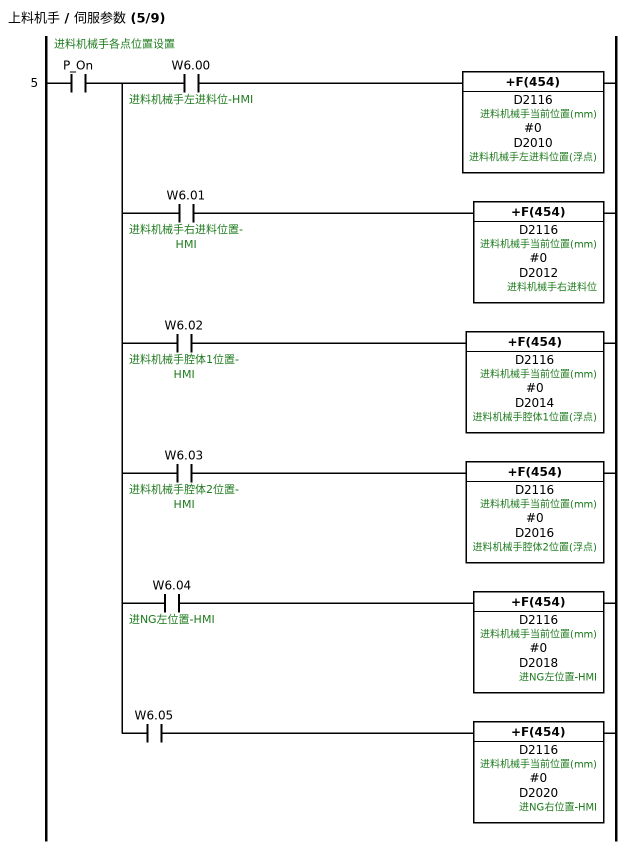
; [picture p96: 上料机手 / 伺服参数, rungs 5-5]
; rung 5: 进料机械手各点位置设置
LD P_On
OUT TR0
AND W6.00  ; 进料机械手左进料位-HMI
+F(454) D2116 #0 D2010  ; 进料机械手当前位置(mm), 进料机械手左进料位置(浮点)
LD TR0
AND W6.01  ; 进料机械手右进料位置-HMI
+F(454) D2116 #0 D2012  ; 进料机械手当前位置(mm), 进料机械手右进料位
LD TR0
AND W6.02  ; 进料机械手腔体1位置-HMI
+F(454) D2116 #0 D2014  ; 进料机械手当前位置(mm), 进料机械手腔体1位置(浮点)
LD TR0
AND W6.03  ; 进料机械手腔体2位置-HMI
+F(454) D2116 #0 D2016  ; 进料机械手当前位置(mm), 进料机械手腔体2位置(浮点)
LD TR0
AND W6.04  ; 进NG左位置-HMI
+F(454) D2116 #0 D2018  ; 进料机械手当前位置(mm), 进NG左位置-HMI
LD TR0
AND W6.05
+F(454) D2116 #0 D2020  ; 进料机械手当前位置(mm), 进NG右位置-HMI

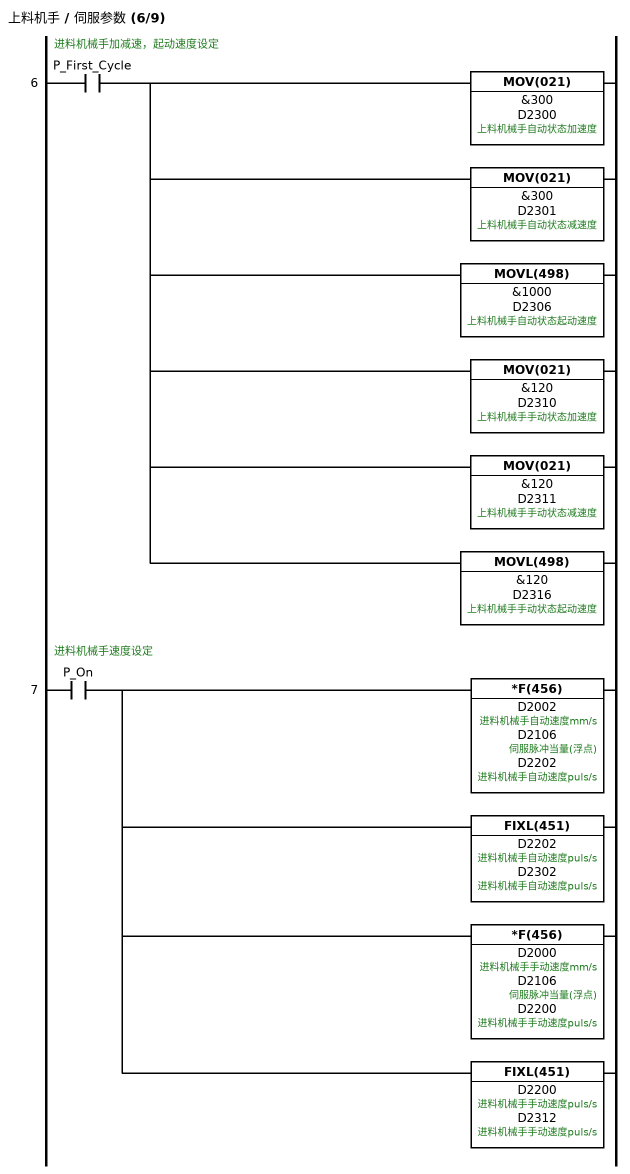
; rung 6: 进料机械手加减速，起动速度设定
LD P_First_Cycle
MOV(021) &300 D2300  ; 上料机械手自动状态加速度
MOV(021) &300 D2301  ; 上料机械手自动状态减速度
MOVL(498) &1000 D2306  ; 上料机械手自动状态起动速度
MOV(021) &120 D2310  ; 上料机械手手动状态加速度
MOV(021) &120 D2311  ; 上料机械手手动状态减速度
MOVL(498) &120 D2316  ; 上料机械手手动状态起动速度
; rung 7: 进料机械手速度设定
LD P_On
*F(456) D2002 D2106 D2202  ; 进料机械手自动速度mm/s, 伺服脉冲当量(浮点), 进料机械手自动速度puls/s
FIXL(451) D2202 D2302  ; 进料机械手自动速度puls/s
*F(456) D2000 D2106 D2200  ; 进料机械手手动速度mm/s, 伺服脉冲当量(浮点), 进料机械手手动速度puls/s
FIXL(451) D2200 D2312  ; 进料机械手手动速度puls/s

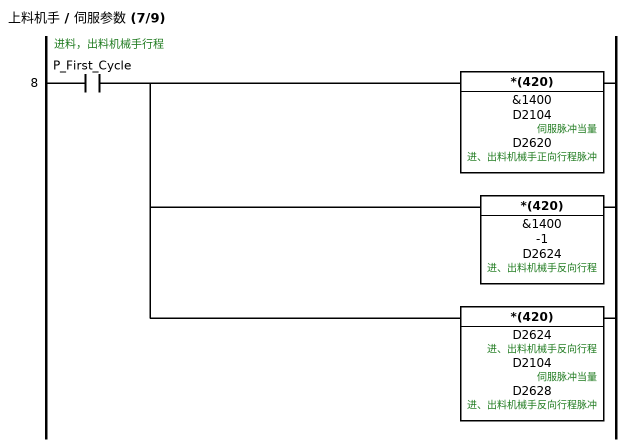
; rung 8: 进料，出料机械手行程
LD P_First_Cycle
*(420) &1400 D2104 D2620  ; 伺服脉冲当量, 进、出料机械手正向行程脉冲
*(420) &1400 -1 D2624  ; 进、出料机械手反向行程
*(420) D2624 D2104 D2628  ; 进、出料机械手反向行程, 伺服脉冲当量, 进、出料机械手反向行程脉冲

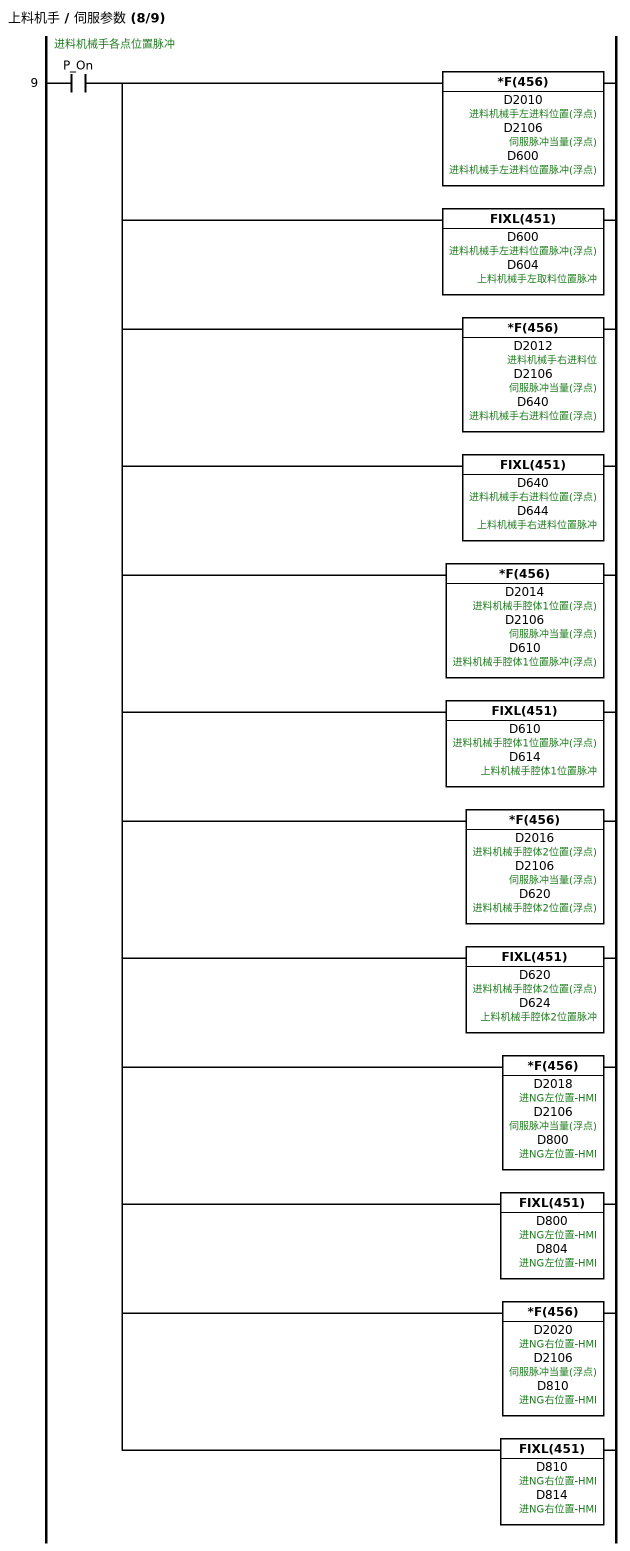
; rung 9: 进料机械手各点位置脉冲
LD P_On
*F(456) D2010 D2106 D600  ; 进料机械手左进料位置(浮点), 伺服脉冲当量(浮点), 进料机械手左进料位置脉冲(浮点)
FIXL(451) D600 D604  ; 进料机械手左进料位置脉冲(浮点), 上料机械手左取料位置脉冲
*F(456) D2012 D2106 D640  ; 进料机械手右进料位, 伺服脉冲当量(浮点), 进料机械手右进料位置(浮点)
FIXL(451) D640 D644  ; 进料机械手右进料位置(浮点), 上料机械手右进料位置脉冲
*F(456) D2014 D2106 D610  ; 进料机械手腔体1位置(浮点), 伺服脉冲当量(浮点), 进料机械手腔体1位置脉冲(浮点)
FIXL(451) D610 D614  ; 进料机械手腔体1位置脉冲(浮点), 上料机械手腔体1位置脉冲
*F(456) D2016 D2106 D620  ; 进料机械手腔体2位置(浮点), 伺服脉冲当量(浮点)
FIXL(451) D620 D624  ; 进料机械手腔体2位置(浮点), 上料机械手腔体2位置脉冲
*F(456) D2018 D2106 D800  ; 进NG左位置-HMI, 伺服脉冲当量(浮点)
FIXL(451) D800 D804  ; 进NG左位置-HMI
*F(456) D2020 D2106 D810  ; 进NG右位置-HMI, 伺服脉冲当量(浮点)
FIXL(451) D810 D814  ; 进NG右位置-HMI

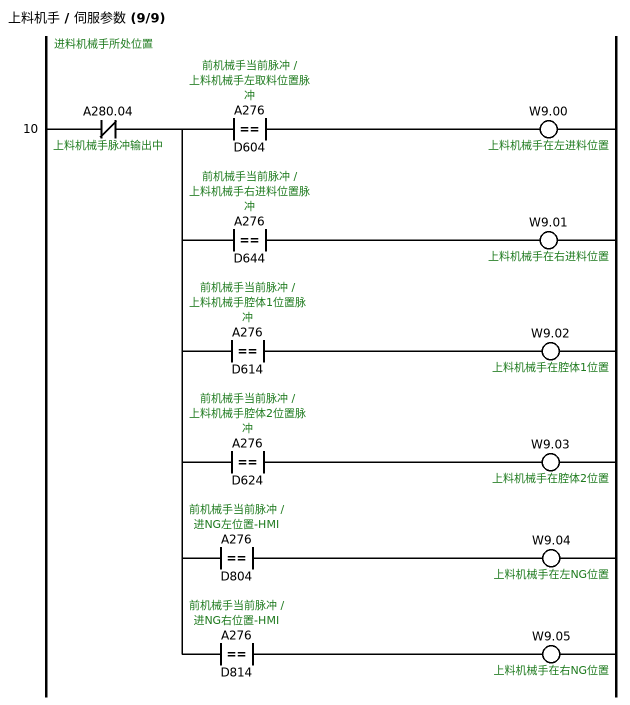
; rung 10: 进料机械手所处位置
LDNOT A280.04  ; 上料机械手脉冲输出中
OUT TR0
AND=SL(303) A276 D604  ; 前机械手当前脉冲, 上料机械手左取料位置脉冲
OUT W9.00  ; 上料机械手在左进料位置
LD TR0
AND=SL(303) A276 D644  ; 前机械手当前脉冲, 上料机械手右进料位置脉冲
OUT W9.01  ; 上料机械手在右进料位置
LD TR0
AND=SL(303) A276 D614  ; 前机械手当前脉冲, 上料机械手腔体1位置脉冲
OUT W9.02  ; 上料机械手在腔体1位置
LD TR0
AND=SL(303) A276 D624  ; 前机械手当前脉冲, 上料机械手腔体2位置脉冲
OUT W9.03  ; 上料机械手在腔体2位置
LD TR0
AND=SL(303) A276 D804  ; 前机械手当前脉冲, 进NG左位置-HMI
OUT W9.04  ; 上料机械手在左NG位置
LD TR0
AND=SL(303) A276 D814  ; 前机械手当前脉冲, 进NG右位置-HMI
OUT W9.05  ; 上料机械手在右NG位置

### Section 外部输出及轴控运动

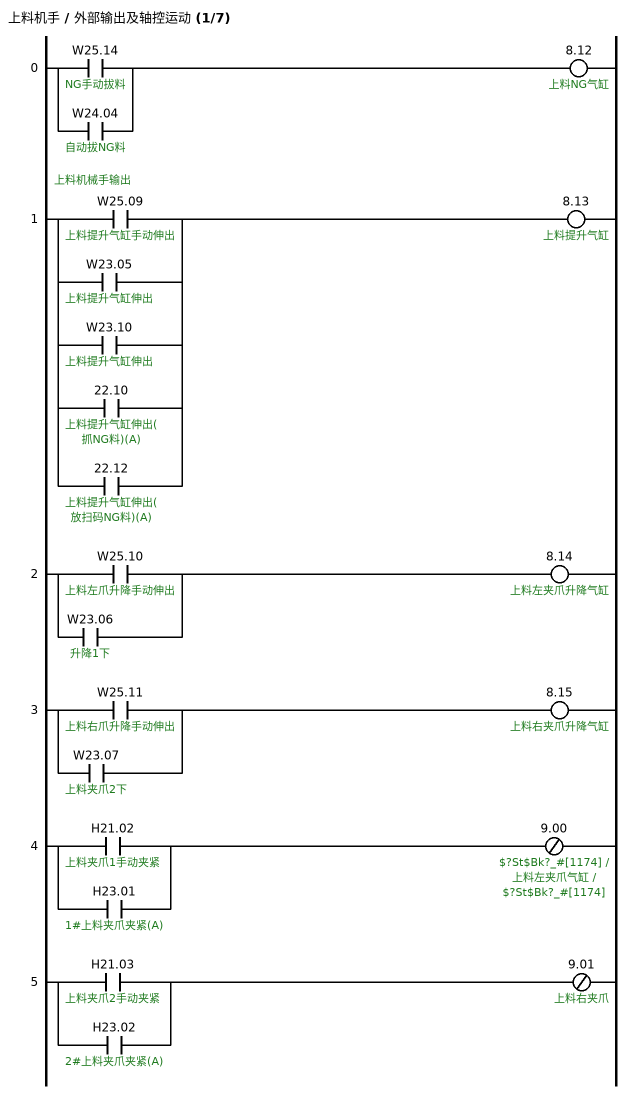
; rung 0
LD W25.14  ; NG手动拔料
OR W24.04  ; 自动拔NG料
OUT 8.12  ; 上料NG气缸
; rung 1: 上料机械手输出
LD W25.09  ; 上料提升气缸手动伸出
OR W23.05  ; 上料提升气缸伸出
OR W23.10  ; 上料提升气缸伸出
OR 22.10  ; 上料提升气缸伸出(抓NG料)(A)
OR 22.12  ; 上料提升气缸伸出(放扫码NG料)(A)
OUT 8.13  ; 上料提升气缸
; rung 2
LD W25.10  ; 上料左爪升降手动伸出
OR W23.06  ; 升降1下
OUT 8.14  ; 上料左夹爪升降气缸
; rung 3
LD W25.11  ; 上料右爪升降手动伸出
OR W23.07  ; 上料夹爪2下
OUT 8.15  ; 上料右夹爪升降气缸
; rung 4
LD H21.02  ; 上料夹爪1手动夹紧
OR H23.01  ; 1#上料夹爪夹紧(A)
OUTNOT 9.00  ; $?St$Bk?_#[1174] / 上料左夹爪气缸 / $?St$Bk?_#[1174]
; rung 5
LD H21.03  ; 上料夹爪2手动夹紧
OR H23.02  ; 2#上料夹爪夹紧(A)
OUTNOT 9.01  ; 上料右夹爪

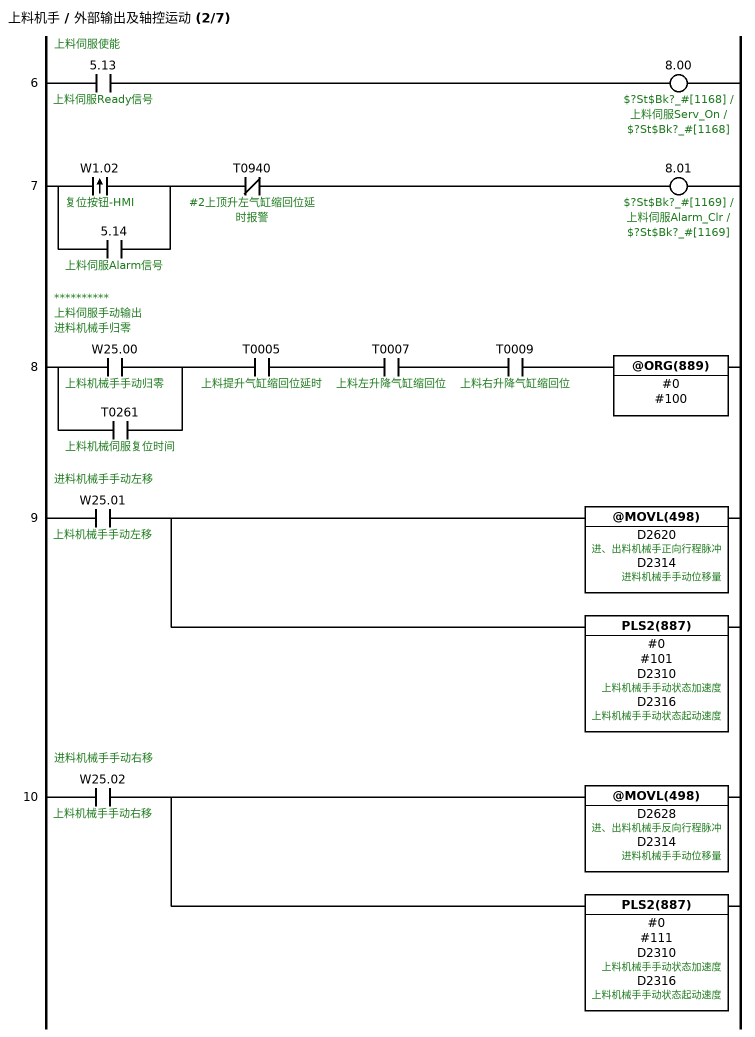
; rung 6: 上料伺服使能
LD 5.13  ; 上料伺服Ready信号
OUT 8.00  ; $?St$Bk?_#[1168] / 上料伺服Serv_On / $?St$Bk?_#[1168]
; rung 7
@LD W1.02  ; 复位按钮-HMI
OR 5.14  ; 上料伺服Alarm信号
ANDNOT T0940  ; #2上顶升左气缸缩回位延时报警
OUT 8.01  ; $?St$Bk?_#[1169] / 上料伺服Alarm_Clr / $?St$Bk?_#[1169]
; rung 8: ********** / 上料伺服手动输出 / 进料机械手归零
LD W25.00  ; 上料机械手手动归零
OR T0261  ; 上料机械伺服复位时间
AND T0005  ; 上料提升气缸缩回位延时
AND T0007  ; 上料左升降气缸缩回位
AND T0009  ; 上料右升降气缸缩回位
@ORG(889) #0 #100
; rung 9: 进料机械手手动左移
LD W25.01  ; 上料机械手手动左移
@MOVL(498) D2620 D2314  ; 进、出料机械手正向行程脉冲, 进料机械手手动位移量
PLS2(887) #0 #101 D2310 D2316  ; 上料机械手手动状态加速度, 上料机械手手动状态起动速度
; rung 10: 进料机械手手动右移
LD W25.02  ; 上料机械手手动右移
@MOVL(498) D2628 D2314  ; 进、出料机械手反向行程脉冲, 进料机械手手动位移量
PLS2(887) #0 #111 D2310 D2316  ; 上料机械手手动状态加速度, 上料机械手手动状态起动速度

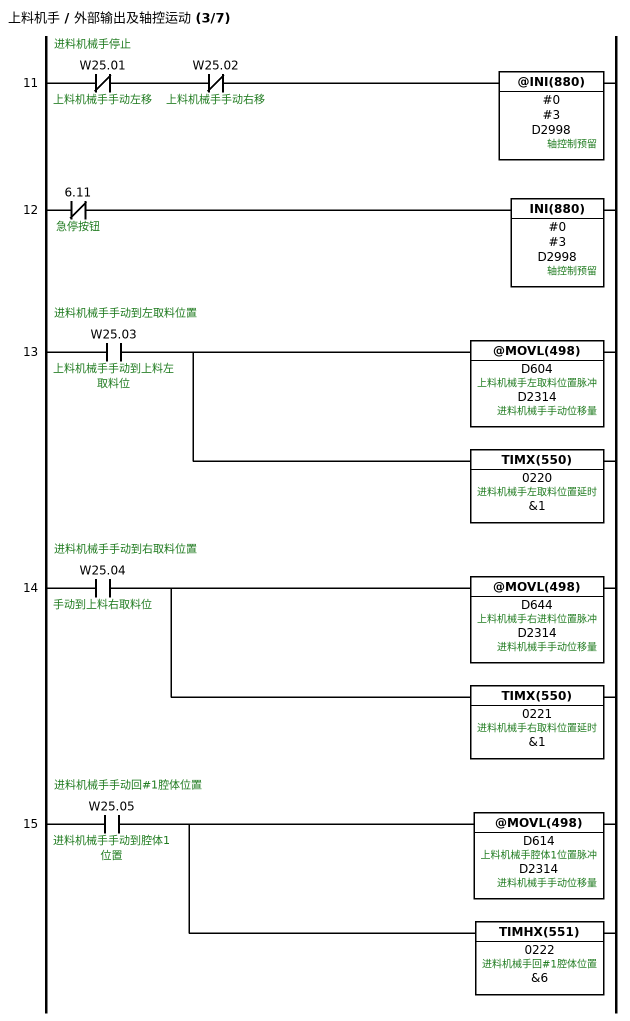
; rung 11: 进料机械手停止
LDNOT W25.01  ; 上料机械手手动左移
ANDNOT W25.02  ; 上料机械手手动右移
@INI(880) #0 #3 D2998  ; 轴控制预留
; rung 12
LDNOT 6.11  ; 急停按钮
INI(880) #0 #3 D2998  ; 轴控制预留
; rung 13: 进料机械手手动到左取料位置
LD W25.03  ; 上料机械手手动到上料左取料位
@MOVL(498) D604 D2314  ; 上料机械手左取料位置脉冲, 进料机械手手动位移量
TIMX(550) 0220 &1  ; 进料机械手左取料位置延时
; rung 14: 进料机械手手动到右取料位置
LD W25.04  ; 手动到上料右取料位
@MOVL(498) D644 D2314  ; 上料机械手右进料位置脉冲, 进料机械手手动位移量
TIMX(550) 0221 &1  ; 进料机械手右取料位置延时
; rung 15: 进料机械手手动回#1腔体位置
LD W25.05  ; 进料机械手手动到腔体1位置
@MOVL(498) D614 D2314  ; 上料机械手腔体1位置脉冲, 进料机械手手动位移量
TIMHX(551) 0222 &6  ; 进料机械手回#1腔体位置

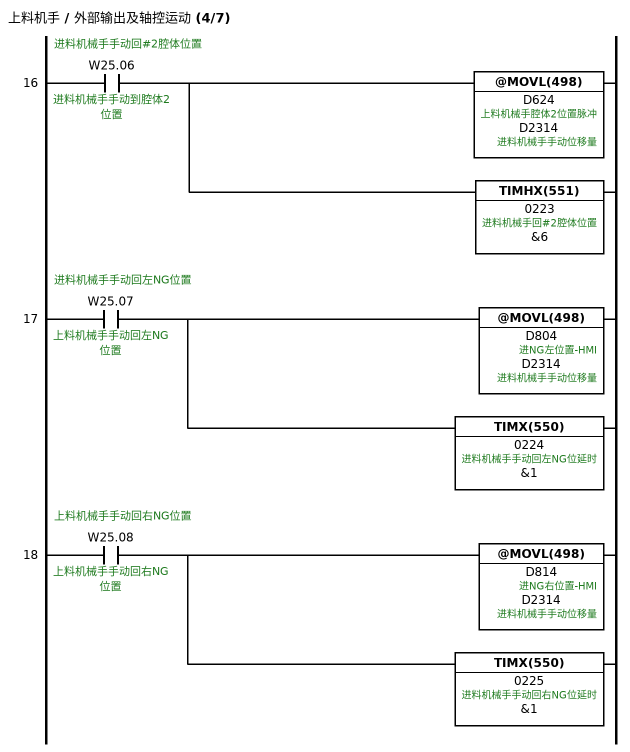
; rung 16: 进料机械手手动回#2腔体位置
LD W25.06  ; 进料机械手手动到腔体2位置
@MOVL(498) D624 D2314  ; 上料机械手腔体2位置脉冲, 进料机械手手动位移量
TIMHX(551) 0223 &6  ; 进料机械手回#2腔体位置
; rung 17: 进料机械手手动回左NG位置
LD W25.07  ; 上料机械手手动回左NG位置
@MOVL(498) D804 D2314  ; 进NG左位置-HMI, 进料机械手手动位移量
TIMX(550) 0224 &1  ; 进料机械手手动回左NG位延时
; rung 18: 上料机械手手动回右NG位置
LD W25.08  ; 上料机械手手动回右NG位置
@MOVL(498) D814 D2314  ; 进NG右位置-HMI, 进料机械手手动位移量
TIMX(550) 0225 &1  ; 进料机械手手动回右NG位延时

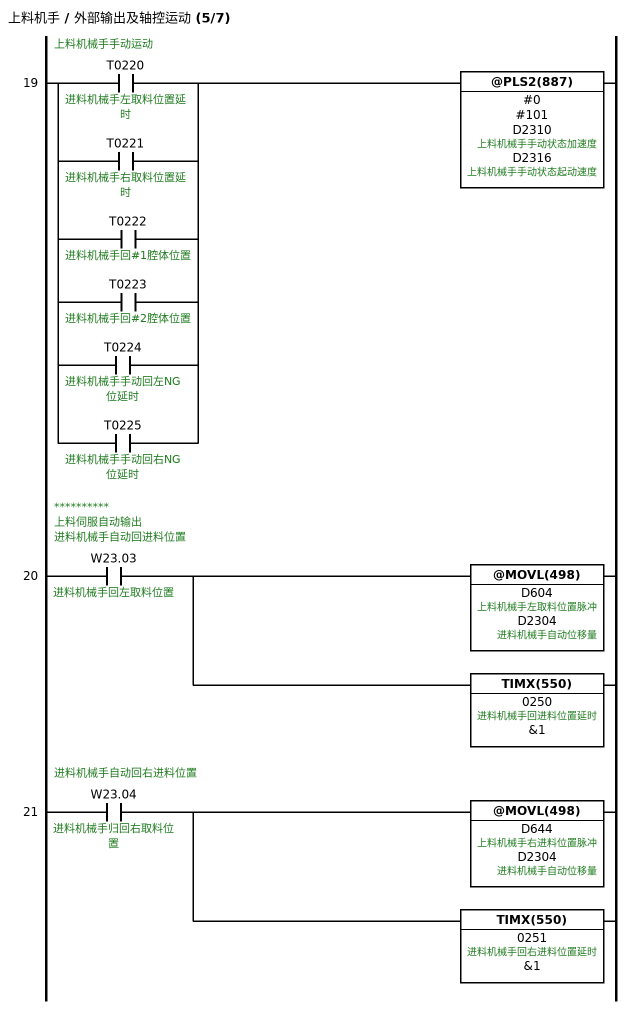
; rung 19: 上料机械手手动运动
LD T0220  ; 进料机械手左取料位置延时
OR T0221  ; 进料机械手右取料位置延时
OR T0222  ; 进料机械手回#1腔体位置
OR T0223  ; 进料机械手回#2腔体位置
OR T0224  ; 进料机械手手动回左NG位延时
OR T0225  ; 进料机械手手动回右NG位延时
@PLS2(887) #0 #101 D2310 D2316  ; 上料机械手手动状态加速度, 上料机械手手动状态起动速度
; rung 20: ********** / 上料伺服自动输出 / 进料机械手自动回进料位置
LD W23.03  ; 进料机械手回左取料位置
@MOVL(498) D604 D2304  ; 上料机械手左取料位置脉冲, 进料机械手自动位移量
TIMX(550) 0250 &1  ; 进料机械手回进料位置延时
; rung 21: 进料机械手自动回右进料位置
LD W23.04  ; 进料机械手归回右取料位置
@MOVL(498) D644 D2304  ; 上料机械手右进料位置脉冲, 进料机械手自动位移量
TIMX(550) 0251 &1  ; 进料机械手回右进料位置延时

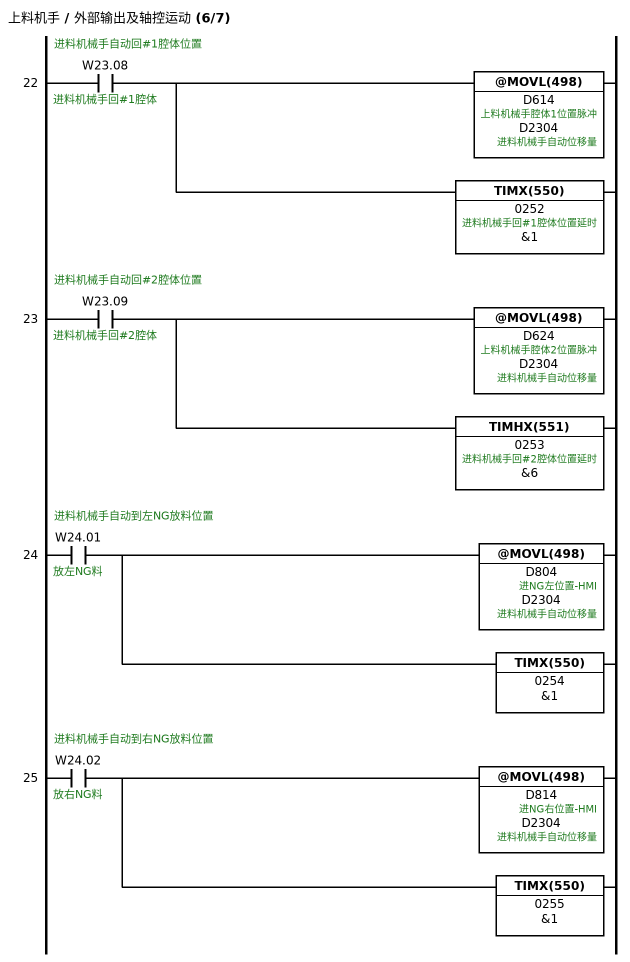
; rung 22: 进料机械手自动回#1腔体位置
LD W23.08  ; 进料机械手回#1腔体
@MOVL(498) D614 D2304  ; 上料机械手腔体1位置脉冲, 进料机械手自动位移量
TIMX(550) 0252 &1  ; 进料机械手回#1腔体位置延时
; rung 23: 进料机械手自动回#2腔体位置
LD W23.09  ; 进料机械手回#2腔体
@MOVL(498) D624 D2304  ; 上料机械手腔体2位置脉冲, 进料机械手自动位移量
TIMHX(551) 0253 &6  ; 进料机械手回#2腔体位置延时
; rung 24: 进料机械手自动到左NG放料位置
LD W24.01  ; 放左NG料
@MOVL(498) D804 D2304  ; 进NG左位置-HMI, 进料机械手自动位移量
TIMX(550) 0254 &1
; rung 25: 进料机械手自动到右NG放料位置
LD W24.02  ; 放右NG料
@MOVL(498) D814 D2304  ; 进NG右位置-HMI, 进料机械手自动位移量
TIMX(550) 0255 &1

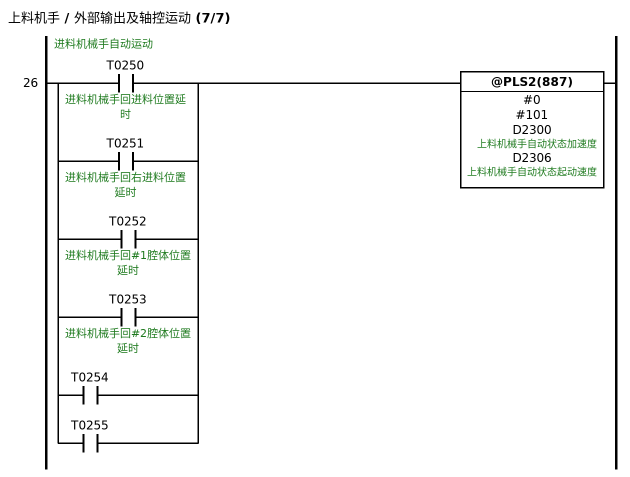
; rung 26: 进料机械手自动运动
LD T0250  ; 进料机械手回进料位置延时
OR T0251  ; 进料机械手回右进料位置延时
OR T0252  ; 进料机械手回#1腔体位置延时
OR T0253  ; 进料机械手回#2腔体位置延时
OR T0254
OR T0255
@PLS2(887) #0 #101 D2300 D2306  ; 上料机械手自动状态加速度, 上料机械手自动状态起动速度

### Section 自动报警

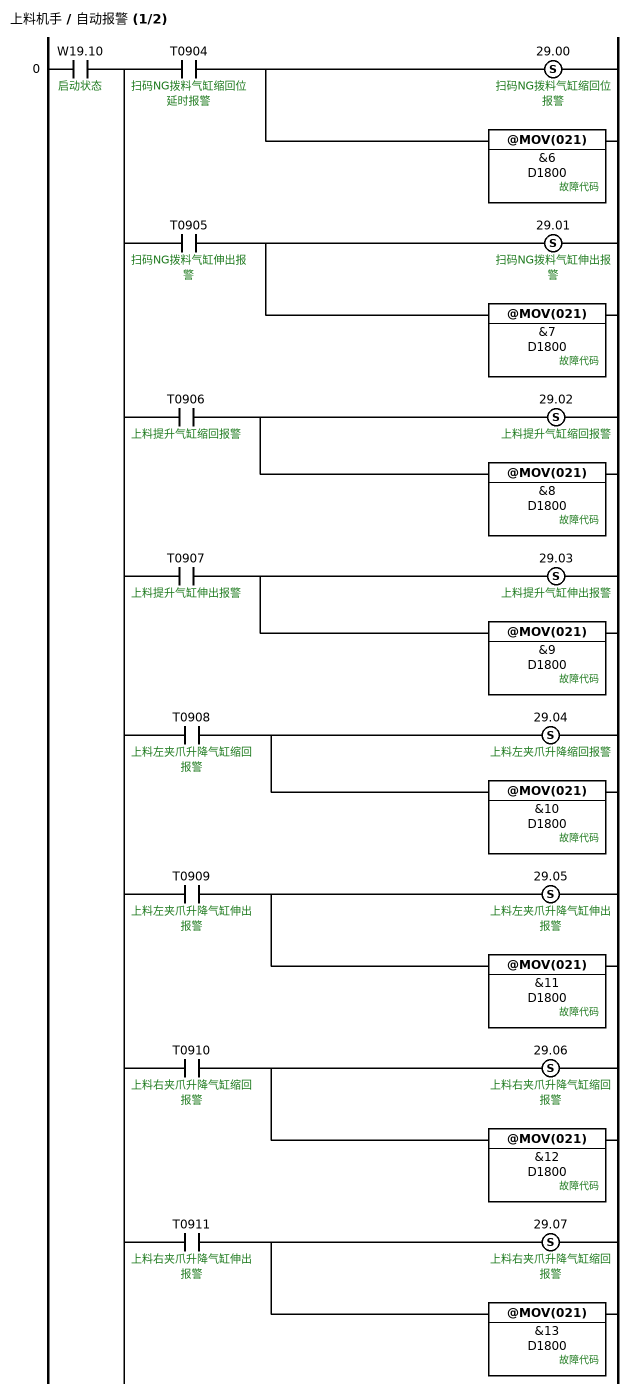

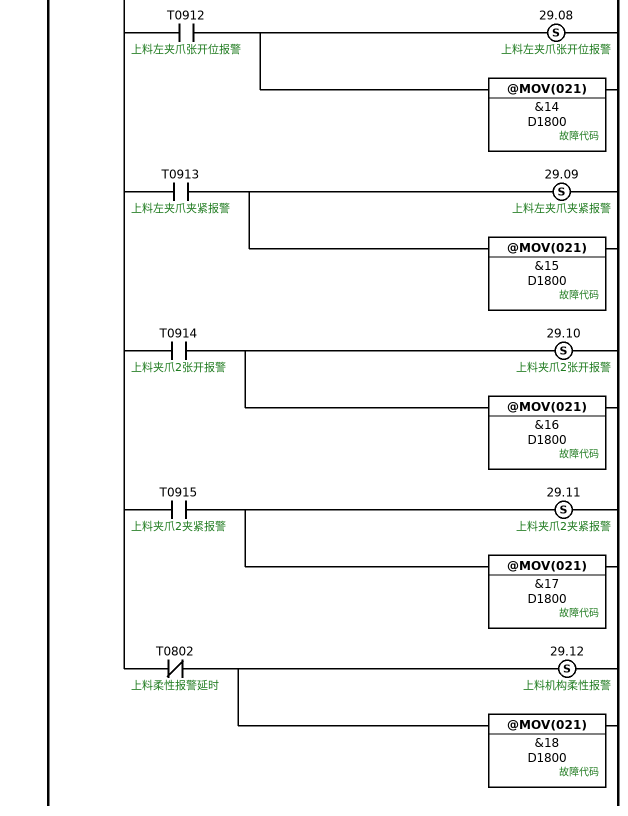
; rung 0
LD W19.10  ; 启动状态
OUT TR0
AND T0904  ; 扫码NG拨料气缸缩回位延时报警
SET 29.00  ; 扫码NG拨料气缸缩回位报警
@MOV(021) &6 D1800  ; 故障代码
LD TR0
AND T0905  ; 扫码NG拨料气缸伸出报警
SET 29.01  ; 扫码NG拨料气缸伸出报警
@MOV(021) &7 D1800  ; 故障代码
LD TR0
AND T0906  ; 上料提升气缸缩回报警
SET 29.02  ; 上料提升气缸缩回报警
@MOV(021) &8 D1800  ; 故障代码
LD TR0
AND T0907  ; 上料提升气缸伸出报警
SET 29.03  ; 上料提升气缸伸出报警
@MOV(021) &9 D1800  ; 故障代码
LD TR0
AND T0908  ; 上料左夹爪升降气缸缩回报警
SET 29.04  ; 上料左夹爪升降缩回报警
@MOV(021) &10 D1800  ; 故障代码
LD TR0
AND T0909  ; 上料左夹爪升降气缸伸出报警
SET 29.05  ; 上料左夹爪升降气缸伸出报警
@MOV(021) &11 D1800  ; 故障代码
LD TR0
AND T0910  ; 上料右夹爪升降气缸缩回报警
SET 29.06  ; 上料右夹爪升降气缸缩回报警
@MOV(021) &12 D1800  ; 故障代码
LD TR0
AND T0911  ; 上料右夹爪升降气缸伸出报警
SET 29.07  ; 上料右夹爪升降气缸缩回报警
@MOV(021) &13 D1800  ; 故障代码
LD TR0
AND T0912  ; 上料左夹爪张开位报警
SET 29.08  ; 上料左夹爪张开位报警
@MOV(021) &14 D1800  ; 故障代码
LD TR0
AND T0913  ; 上料左夹爪夹紧报警
SET 29.09  ; 上料左夹爪夹紧报警
@MOV(021) &15 D1800  ; 故障代码
LD TR0
AND T0914  ; 上料夹爪2张开报警
SET 29.10  ; 上料夹爪2张开报警
@MOV(021) &16 D1800  ; 故障代码
LD TR0
AND T0915  ; 上料夹爪2夹紧报警
SET 29.11  ; 上料夹爪2夹紧报警
@MOV(021) &17 D1800  ; 故障代码
LD TR0
ANDNOT T0802  ; 上料柔性报警延时
SET 29.12  ; 上料机构柔性报警
@MOV(021) &18 D1800  ; 故障代码

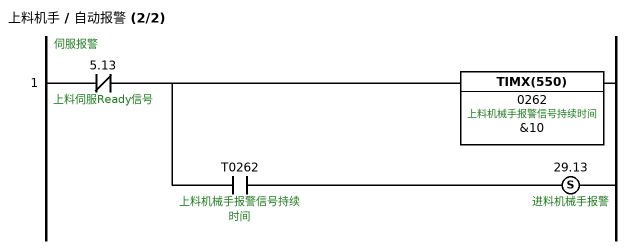
; rung 1: 伺服报警
LDNOT 5.13  ; 上料伺服Ready信号
TIMX(550) 0262 &10  ; 上料机械手报警信号持续时间
AND T0262  ; 上料机械手报警信号持续时间
SET 29.13  ; 进料机械手报警

### Section 上料机械手复位

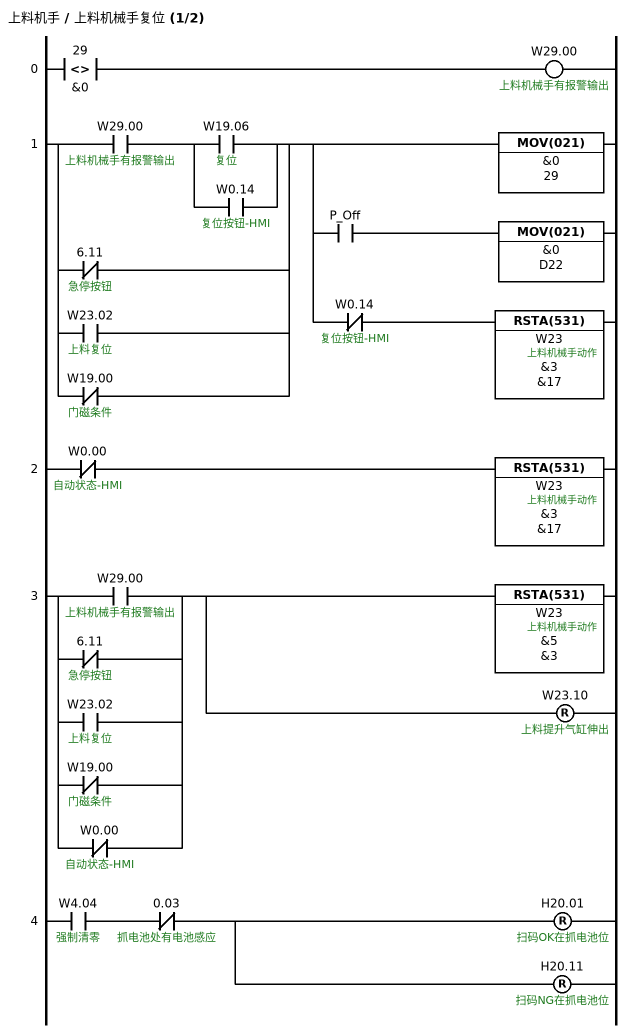
; rung 0
LD<>(305) 29 &0
OUT W29.00  ; 上料机械手有报警输出
; rung 1
LD W29.00  ; 上料机械手有报警输出
LD W19.06  ; 复位
OR W0.14  ; 复位按钮-HMI
ANDLD
ORNOT 6.11  ; 急停按钮
OR W23.02  ; 上料复位
ORNOT W19.00  ; 门磁条件
OUT TR0
MOV(021) &0 29
AND P_Off
MOV(021) &0 D22
LD TR0
ANDNOT W0.14  ; 复位按钮-HMI
RSTA(531) W23 &3 &17  ; 上料机械手动作
; rung 2
LDNOT W0.00  ; 自动状态-HMI
RSTA(531) W23 &3 &17  ; 上料机械手动作
; rung 3
LD W29.00  ; 上料机械手有报警输出
ORNOT 6.11  ; 急停按钮
OR W23.02  ; 上料复位
ORNOT W19.00  ; 门磁条件
ORNOT W0.00  ; 自动状态-HMI
RSTA(531) W23 &5 &3  ; 上料机械手动作
RSET W23.10  ; 上料提升气缸伸出
; rung 4
LD W4.04  ; 强制清零
ANDNOT 0.03  ; 抓电池处有电池感应
RSET H20.01  ; 扫码OK在抓电池位
RSET H20.11  ; 扫码NG在抓电池位

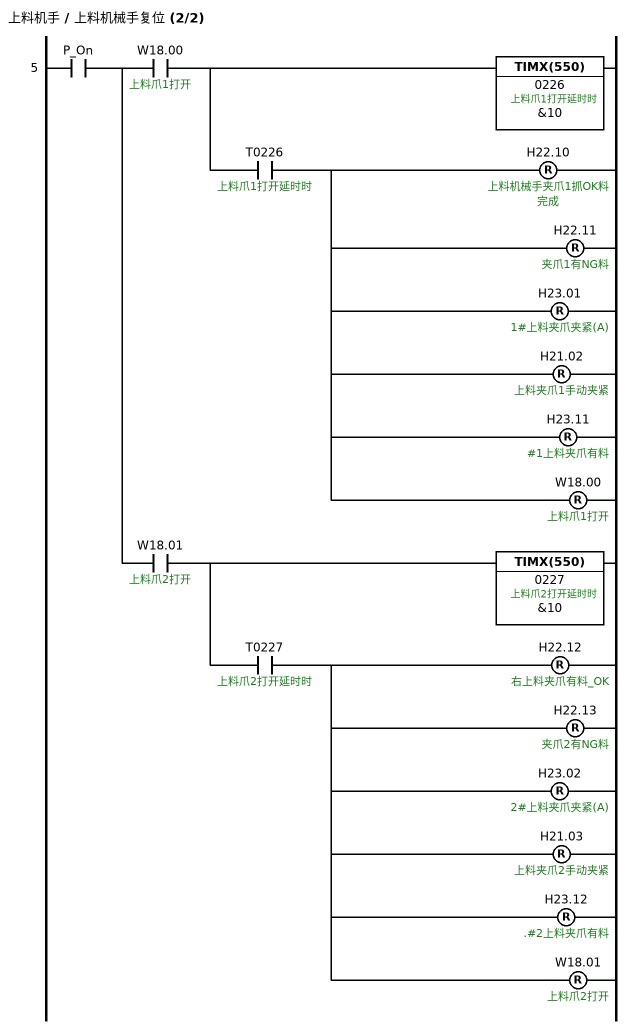
; rung 5
LD P_On
OUT TR0
AND W18.00  ; 上料爪1打开
TIMX(550) 0226 &10  ; 上料爪1打开延时时
AND T0226  ; 上料爪1打开延时时
RSET H22.10  ; 上料机械手夹爪1抓OK料完成
RSET H22.11  ; 夹爪1有NG料
RSET H23.01  ; 1#上料夹爪夹紧(A)
RSET H21.02  ; 上料夹爪1手动夹紧
RSET H23.11  ; #1上料夹爪有料
RSET W18.00  ; 上料爪1打开
LD TR0
AND W18.01  ; 上料爪2打开
TIMX(550) 0227 &10  ; 上料爪2打开延时时
AND T0227  ; 上料爪2打开延时时
RSET H22.12  ; 右上料夹爪有料_OK
RSET H22.13  ; 夹爪2有NG料
RSET H23.02  ; 2#上料夹爪夹紧(A)
RSET H21.03  ; 上料夹爪2手动夹紧
RSET H23.12  ; .#2上料夹爪有料
RSET W18.01  ; 上料爪2打开

### Section END
; rung 0
END(001)

## Program 测试腔体 (cyclic task 3)

### Section 腔体1手动

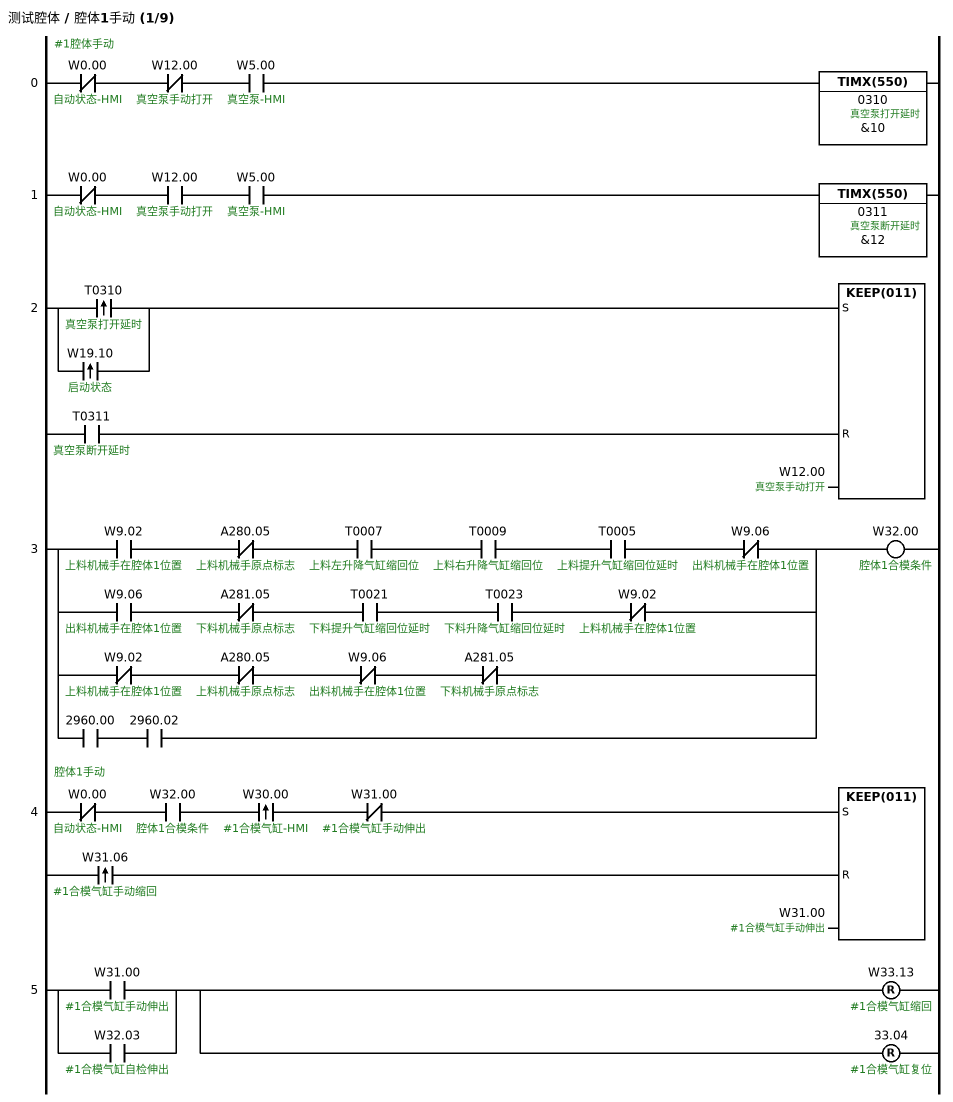
; rung 0: #1腔体手动
LDNOT W0.00  ; 自动状态-HMI
ANDNOT W12.00  ; 真空泵手动打开
AND W5.00  ; 真空泵-HMI
TIMX(550) 0310 &10  ; 真空泵打开延时
; rung 1
LDNOT W0.00  ; 自动状态-HMI
AND W12.00  ; 真空泵手动打开
AND W5.00  ; 真空泵-HMI
TIMX(550) 0311 &12  ; 真空泵断开延时
; rung 2
@LD T0310  ; 真空泵打开延时
@OR W19.10  ; 启动状态
LD T0311  ; 真空泵断开延时
KEEP(011) W12.00  ; 真空泵手动打开
; rung 3
LD W9.02  ; 上料机械手在腔体1位置
ANDNOT A280.05  ; 上料机械手原点标志
AND T0007  ; 上料左升降气缸缩回位
AND T0009  ; 上料右升降气缸缩回位
AND T0005  ; 上料提升气缸缩回位延时
ANDNOT W9.06  ; 出料机械手在腔体1位置
LD W9.06  ; 出料机械手在腔体1位置
ANDNOT A281.05  ; 下料机械手原点标志
AND T0021  ; 下料提升气缸缩回位延时
AND T0023  ; 下料升降气缸缩回位延时
ANDNOT W9.02  ; 上料机械手在腔体1位置
ORLD
LDNOT W9.02  ; 上料机械手在腔体1位置
ANDNOT A280.05  ; 上料机械手原点标志
ANDNOT W9.06  ; 出料机械手在腔体1位置
ANDNOT A281.05  ; 下料机械手原点标志
ORLD
LD 2960.00
AND 2960.02
ORLD
OUT W32.00  ; 腔体1合模条件
; rung 4: 腔体1手动
LDNOT W0.00  ; 自动状态-HMI
AND W32.00  ; 腔体1合模条件
@AND W30.00  ; #1合模气缸-HMI
ANDNOT W31.00  ; #1合模气缸手动伸出
@LD W31.06  ; #1合模气缸手动缩回
KEEP(011) W31.00  ; #1合模气缸手动伸出
; rung 5
LD W31.00  ; #1合模气缸手动伸出
OR W32.03  ; #1合模气缸自检伸出
RSET W33.13  ; #1合模气缸缩回
RSET 33.04  ; #1合模气缸复位

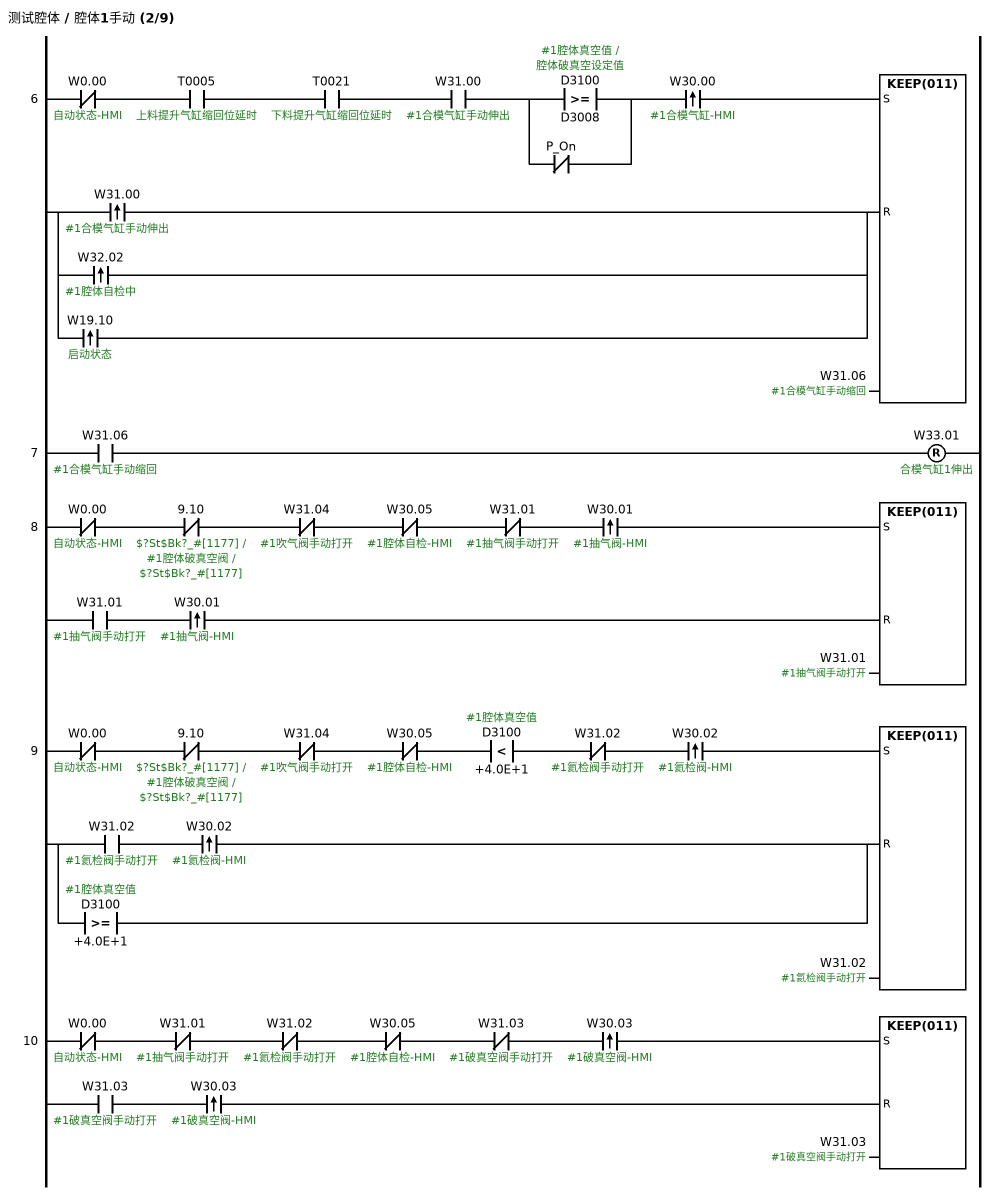
; rung 6
LDNOT W0.00  ; 自动状态-HMI
AND T0005  ; 上料提升气缸缩回位延时
AND T0021  ; 下料提升气缸缩回位延时
AND W31.00  ; #1合模气缸手动伸出
LD>=F(334) D3100 D3008  ; #1腔体真空值, 腔体破真空设定值
ORNOT P_On
ANDLD
@AND W30.00  ; #1合模气缸-HMI
@LD W31.00  ; #1合模气缸手动伸出
@OR W32.02  ; #1腔体自检中
@OR W19.10  ; 启动状态
KEEP(011) W31.06  ; #1合模气缸手动缩回
; rung 7
LD W31.06  ; #1合模气缸手动缩回
RSET W33.01  ; 合模气缸1伸出
; rung 8
LDNOT W0.00  ; 自动状态-HMI
ANDNOT 9.10  ; $?St$Bk?_#[1177] / #1腔体破真空阀 / $?St$Bk?_#[1177]
ANDNOT W31.04  ; #1吹气阀手动打开
ANDNOT W30.05  ; #1腔体自检-HMI
ANDNOT W31.01  ; #1抽气阀手动打开
@AND W30.01  ; #1抽气阀-HMI
LD W31.01  ; #1抽气阀手动打开
@AND W30.01  ; #1抽气阀-HMI
KEEP(011) W31.01  ; #1抽气阀手动打开
; rung 9
LDNOT W0.00  ; 自动状态-HMI
ANDNOT 9.10  ; $?St$Bk?_#[1177] / #1腔体破真空阀 / $?St$Bk?_#[1177]
ANDNOT W31.04  ; #1吹气阀手动打开
ANDNOT W30.05  ; #1腔体自检-HMI
AND<F(331) D3100 +4.0E+1  ; #1腔体真空值
ANDNOT W31.02  ; #1氦检阀手动打开
@AND W30.02  ; #1氦检阀-HMI
LD W31.02  ; #1氦检阀手动打开
@AND W30.02  ; #1氦检阀-HMI
OR>=F(334) D3100 +4.0E+1  ; #1腔体真空值
KEEP(011) W31.02  ; #1氦检阀手动打开
; rung 10
LDNOT W0.00  ; 自动状态-HMI
ANDNOT W31.01  ; #1抽气阀手动打开
ANDNOT W31.02  ; #1氦检阀手动打开
ANDNOT W30.05  ; #1腔体自检-HMI
ANDNOT W31.03  ; #1破真空阀手动打开
@AND W30.03  ; #1破真空阀-HMI
LD W31.03  ; #1破真空阀手动打开
@AND W30.03  ; #1破真空阀-HMI
KEEP(011) W31.03  ; #1破真空阀手动打开

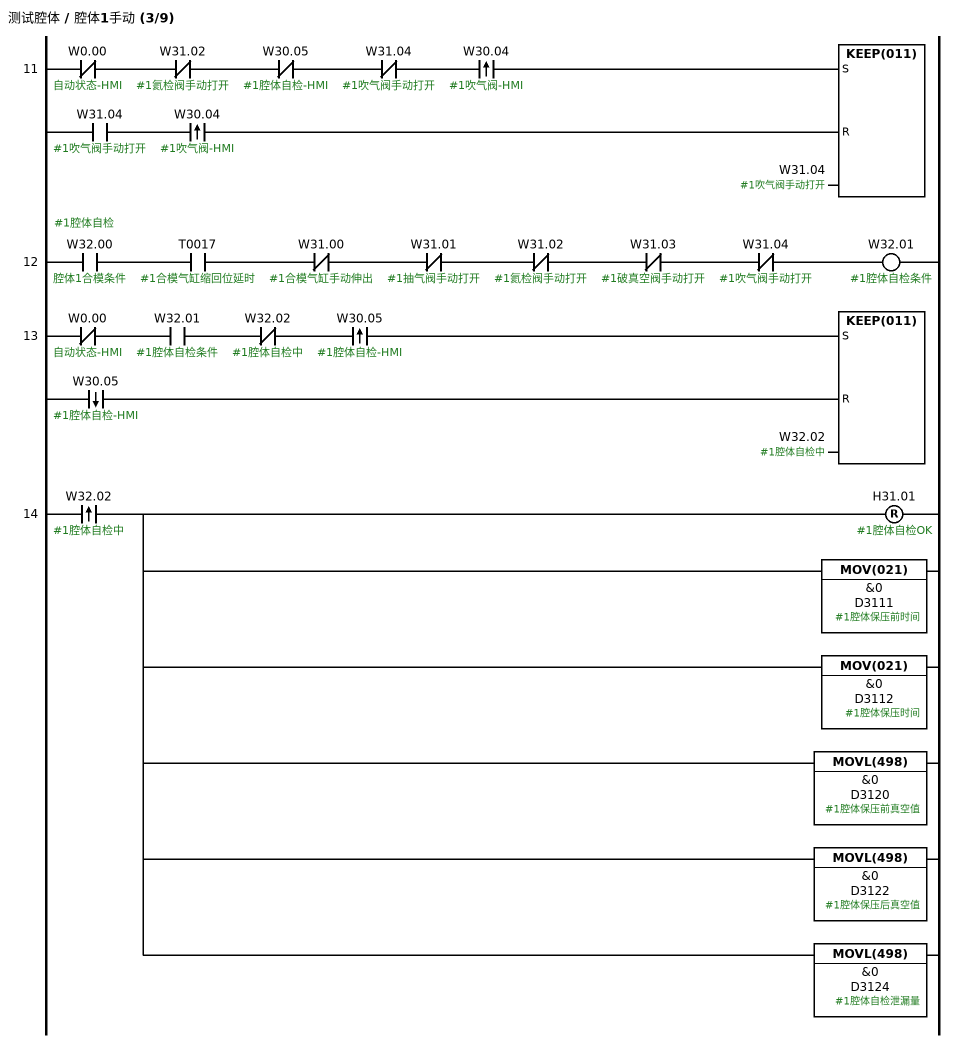
; rung 11
LDNOT W0.00  ; 自动状态-HMI
ANDNOT W31.02  ; #1氦检阀手动打开
ANDNOT W30.05  ; #1腔体自检-HMI
ANDNOT W31.04  ; #1吹气阀手动打开
@AND W30.04  ; #1吹气阀-HMI
LD W31.04  ; #1吹气阀手动打开
@AND W30.04  ; #1吹气阀-HMI
KEEP(011) W31.04  ; #1吹气阀手动打开
; rung 12: #1腔体自检
LD W32.00  ; 腔体1合模条件
AND T0017  ; #1合模气缸缩回位延时
ANDNOT W31.00  ; #1合模气缸手动伸出
ANDNOT W31.01  ; #1抽气阀手动打开
ANDNOT W31.02  ; #1氦检阀手动打开
ANDNOT W31.03  ; #1破真空阀手动打开
ANDNOT W31.04  ; #1吹气阀手动打开
OUT W32.01  ; #1腔体自检条件
; rung 13
LDNOT W0.00  ; 自动状态-HMI
AND W32.01  ; #1腔体自检条件
ANDNOT W32.02  ; #1腔体自检中
@AND W30.05  ; #1腔体自检-HMI
%LD W30.05  ; #1腔体自检-HMI
KEEP(011) W32.02  ; #1腔体自检中
; rung 14
@LD W32.02  ; #1腔体自检中
RSET H31.01  ; #1腔体自检OK
MOV(021) &0 D3111  ; #1腔体保压前时间
MOV(021) &0 D3112  ; #1腔体保压时间
MOVL(498) &0 D3120  ; #1腔体保压前真空值
MOVL(498) &0 D3122  ; #1腔体保压后真空值
MOVL(498) &0 D3124  ; #1腔体自检泄漏量

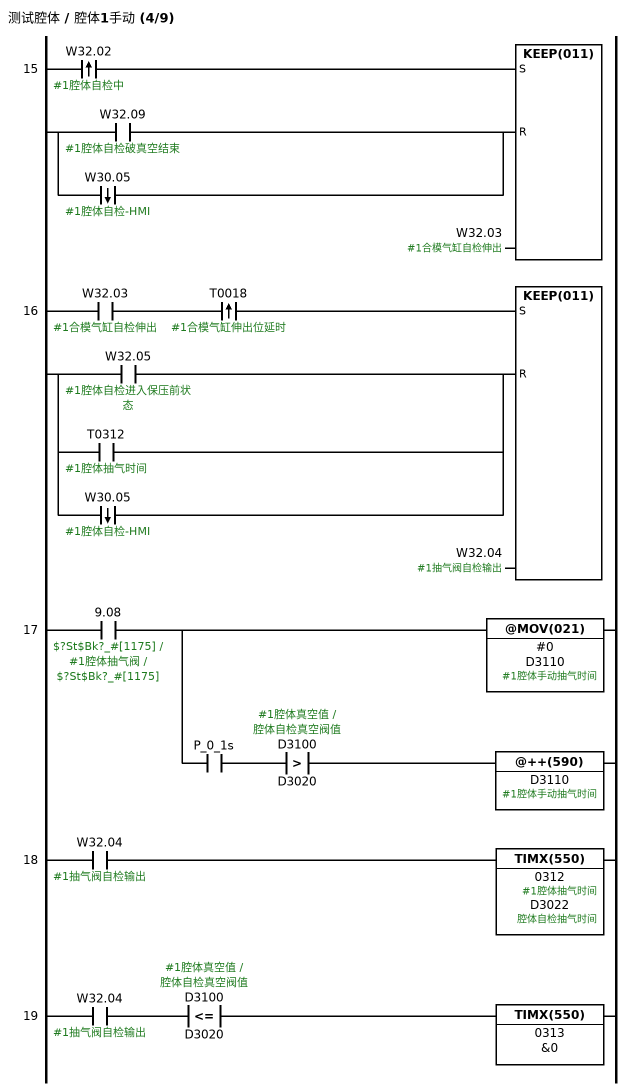
; rung 15
@LD W32.02  ; #1腔体自检中
LD W32.09  ; #1腔体自检破真空结束
%OR W30.05  ; #1腔体自检-HMI
KEEP(011) W32.03  ; #1合模气缸自检伸出
; rung 16
LD W32.03  ; #1合模气缸自检伸出
@AND T0018  ; #1合模气缸伸出位延时
LD W32.05  ; #1腔体自检进入保压前状态
OR T0312  ; #1腔体抽气时间
%OR W30.05  ; #1腔体自检-HMI
KEEP(011) W32.04  ; #1抽气阀自检输出
; rung 17
LD 9.08  ; $?St$Bk?_#[1175] / #1腔体抽气阀 / $?St$Bk?_#[1175]
@MOV(021) #0 D3110  ; #1腔体手动抽气时间
AND P_0_1s
AND>F(333) D3100 D3020  ; #1腔体真空值, 腔体自检真空阀值
@++(590) D3110  ; #1腔体手动抽气时间
; rung 18
LD W32.04  ; #1抽气阀自检输出
TIMX(550) 0312 D3022  ; 腔体自检抽气时间, #1腔体抽气时间
; rung 19
LD W32.04  ; #1抽气阀自检输出
AND<=F(332) D3100 D3020  ; #1腔体真空值, 腔体自检真空阀值
TIMX(550) 0313 &0

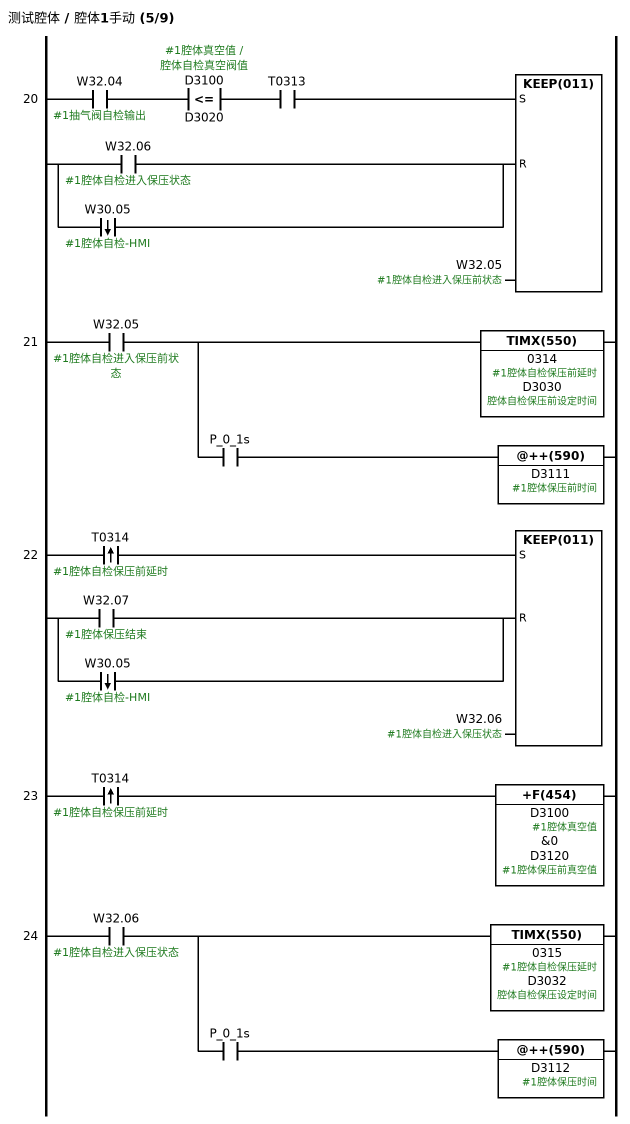
; rung 20
LD W32.04  ; #1抽气阀自检输出
AND<=F(332) D3100 D3020  ; #1腔体真空值, 腔体自检真空阀值
AND T0313
LD W32.06  ; #1腔体自检进入保压状态
%OR W30.05  ; #1腔体自检-HMI
KEEP(011) W32.05  ; #1腔体自检进入保压前状态
; rung 21
LD W32.05  ; #1腔体自检进入保压前状态
TIMX(550) 0314 D3030  ; 腔体自检保压前设定时间, #1腔体自检保压前延时
AND P_0_1s
@++(590) D3111  ; #1腔体保压前时间
; rung 22
@LD T0314  ; #1腔体自检保压前延时
LD W32.07  ; #1腔体保压结束
%OR W30.05  ; #1腔体自检-HMI
KEEP(011) W32.06  ; #1腔体自检进入保压状态
; rung 23
@LD T0314  ; #1腔体自检保压前延时
+F(454) D3100 &0 D3120  ; #1腔体真空值, #1腔体保压前真空值
; rung 24
LD W32.06  ; #1腔体自检进入保压状态
TIMX(550) 0315 D3032  ; 腔体自检保压设定时间, #1腔体自检保压延时
AND P_0_1s
@++(590) D3112  ; #1腔体保压时间

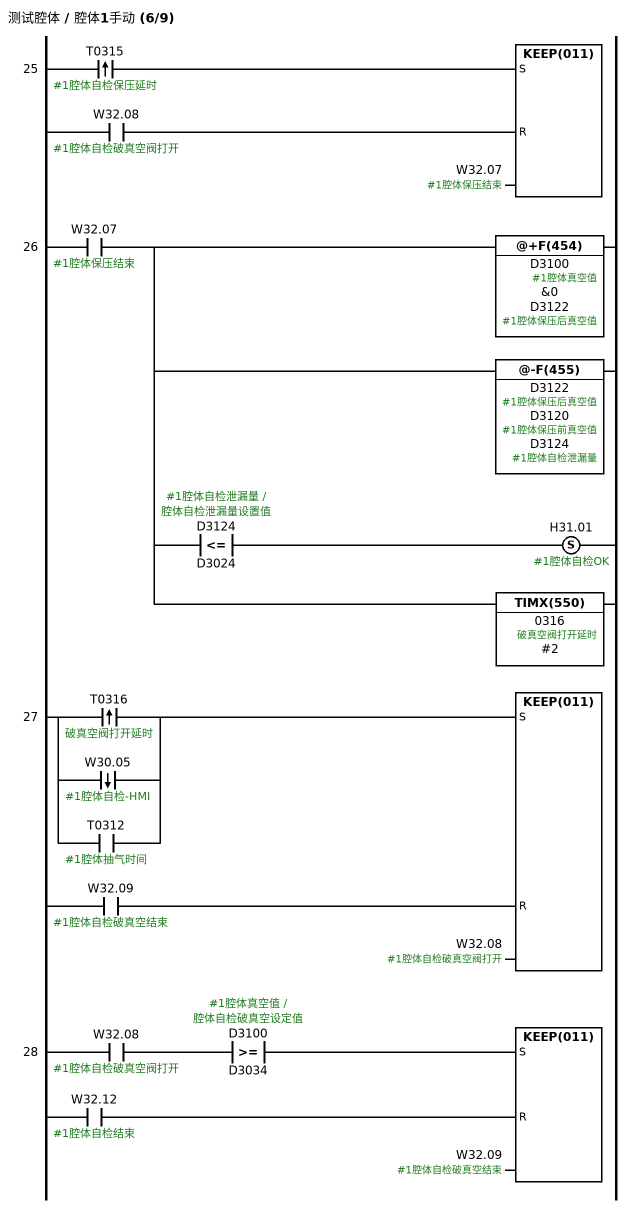
; rung 25
@LD T0315  ; #1腔体自检保压延时
LD W32.08  ; #1腔体自检破真空阀打开
KEEP(011) W32.07  ; #1腔体保压结束
; rung 26
LD W32.07  ; #1腔体保压结束
OUT TR0
@+F(454) D3100 &0 D3122  ; #1腔体真空值, #1腔体保压后真空值
@-F(455) D3122 D3120 D3124  ; #1腔体保压后真空值, #1腔体保压前真空值, #1腔体自检泄漏量
AND<=(315) D3124 D3024  ; #1腔体自检泄漏量, 腔体自检泄漏量设置值
SET H31.01  ; #1腔体自检OK
LD TR0
TIMX(550) 0316 #2  ; 破真空阀打开延时
; rung 27
@LD T0316  ; 破真空阀打开延时
%OR W30.05  ; #1腔体自检-HMI
OR T0312  ; #1腔体抽气时间
LD W32.09  ; #1腔体自检破真空结束
KEEP(011) W32.08  ; #1腔体自检破真空阀打开
; rung 28
LD W32.08  ; #1腔体自检破真空阀打开
AND>=F(334) D3100 D3034  ; #1腔体真空值, 腔体自检破真空设定值
LD W32.12  ; #1腔体自检结束
KEEP(011) W32.09  ; #1腔体自检破真空结束

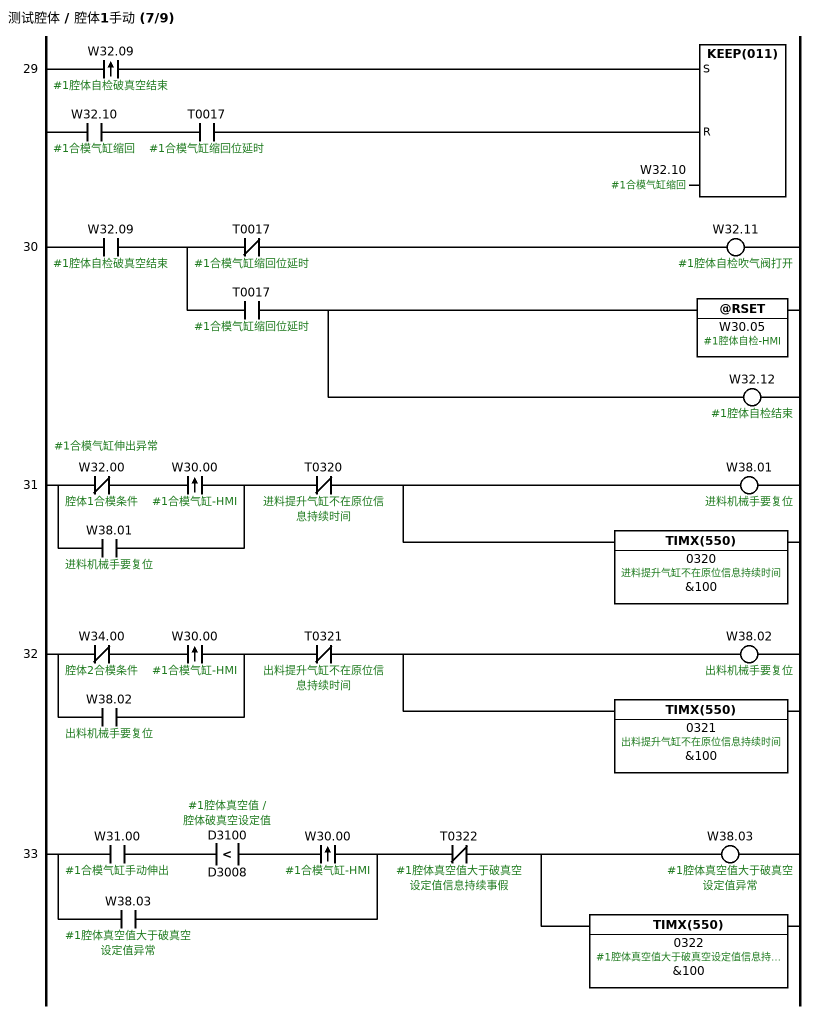
; rung 29
@LD W32.09  ; #1腔体自检破真空结束
LD W32.10  ; #1合模气缸缩回
AND T0017  ; #1合模气缸缩回位延时
KEEP(011) W32.10  ; #1合模气缸缩回
; rung 30
LD W32.09  ; #1腔体自检破真空结束
OUT TR0
ANDNOT T0017  ; #1合模气缸缩回位延时
OUT W32.11  ; #1腔体自检吹气阀打开
LD TR0
AND T0017  ; #1合模气缸缩回位延时
@RSET W30.05  ; #1腔体自检-HMI
OUT W32.12  ; #1腔体自检结束
; rung 31: #1合模气缸伸出异常
LDNOT W32.00  ; 腔体1合模条件
@AND W30.00  ; #1合模气缸-HMI
OR W38.01  ; 进料机械手要复位
ANDNOT T0320  ; 进料提升气缸不在原位信息持续时间
OUT W38.01  ; 进料机械手要复位
TIMX(550) 0320 &100  ; 进料提升气缸不在原位信息持续时间
; rung 32
LDNOT W34.00  ; 腔体2合模条件
@AND W30.00  ; #1合模气缸-HMI
OR W38.02  ; 出料机械手要复位
ANDNOT T0321  ; 出料提升气缸不在原位信息持续时间
OUT W38.02  ; 出料机械手要复位
TIMX(550) 0321 &100  ; 出料提升气缸不在原位信息持续时间
; rung 33
LD W31.00  ; #1合模气缸手动伸出
AND<F(331) D3100 D3008  ; #1腔体真空值, 腔体破真空设定值
@AND W30.00  ; #1合模气缸-HMI
OR W38.03  ; #1腔体真空值大于破真空设定值异常
ANDNOT T0322  ; #1腔体真空值大于破真空设定值信息持续事假
OUT W38.03  ; #1腔体真空值大于破真空设定值异常
TIMX(550) 0322 &100  ; #1腔体真空值大于破真空设定值信息持续事假

